TYPE ST_Order :
STRUCT
	nTargetTable	: INT;
	tWeldingTime	: TIME := T#2S;
	bDone			: BOOL;
	bIsValid		: BOOL;
	bWeld			: BOOL := TRUE;
END_STRUCT
END_TYPE

(* stored: Version 1.1.0.1
   DUT ST_Order: Id {15863fff-617e-48f1-9d77-46ec19d492fa} *)
